(* Logix 5000 project; controller test vendor 1 type 14 code 151 rev 30.11; software revision 30.00 *)

TASK MainTask (continuous, watchdog 500 ms) : MainProgram

MODULES
   Local : vendor 1 type 14 code 151 (Compact 0, rev 30.11)
      Analog_IO : Embedded (Compact 2, rev 1.1, Output RPI 80 ms)
      Discrete_IO : Embedded (Compact 1, rev 3.1, Output RPI 20 ms)
      Counters : Embedded (Compact 3, rev 1.1, Output RPI 20 ms)
END_MODULES

PROGRAM MainProgram   (* main routine MainRoutine *)
VAR
   DI0 : ALIAS FOR Local:1:I.Data.0;
   DI1 : ALIAS FOR Local:1:I.Data.1;
   DI10 : ALIAS FOR Local:1:I.Data.10;
   DI11 : ALIAS FOR Local:1:I.Data.11;
   DI2 : ALIAS FOR Local:1:I.Data.2;
   DI3 : ALIAS FOR Local:1:I.Data.3;
   DI4 : ALIAS FOR Local:1:I.Data.4;
   DI5 : ALIAS FOR Local:1:I.Data.5;
   DI6 : ALIAS FOR Local:1:I.Data.6;
   DI61 : ALIAS FOR Local:1:I.Data.6;
   DI7 : ALIAS FOR Local:1:I.Data.7;
   DI8 : ALIAS FOR Local:1:I.Data.8;
   DI9 : ALIAS FOR Local:1:I.Data.9;
   DO0 : ALIAS FOR Local:1:O.Data.0;
   DO1 : ALIAS FOR Local:1:O.Data.1;
   DO10 : ALIAS FOR Local:1:O.Data.10;
   DO11 : ALIAS FOR Local:1:O.Data.11;
   DO2 : ALIAS FOR Local:1:O.Data.2;
   DO3 : ALIAS FOR Local:1:O.Data.3;
   DO4 : ALIAS FOR Local:1:O.Data.4;
   DO5 : ALIAS FOR Local:1:O.Data.5;
   DO6 : ALIAS FOR Local:1:O.Data.6;
   DO7 : ALIAS FOR Local:1:O.Data.7;
   DO8 : ALIAS FOR Local:1:O.Data.8;
   DO9 : ALIAS FOR Local:1:O.Data.9;
END_VAR

ROUTINE MainRoutine   (* ladder *)
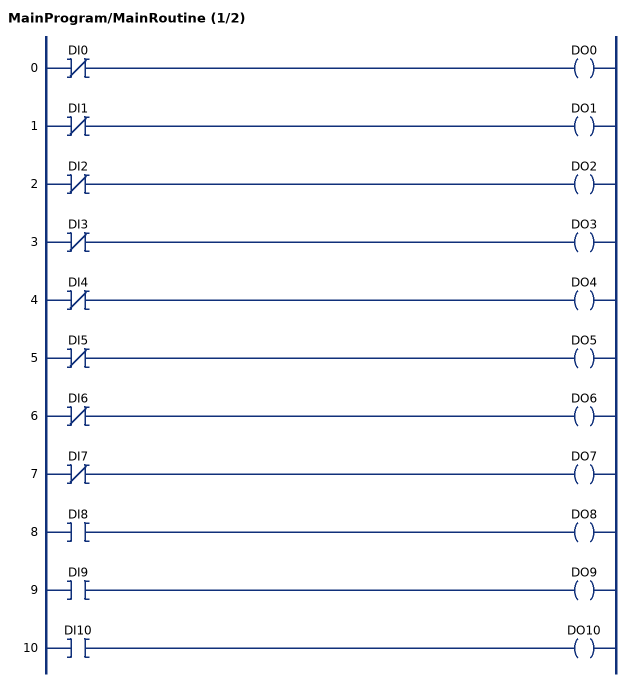
   0: XIO(DI0)OTE(DO0);
   1: XIO(DI1)OTE(DO1);
   2: XIO(DI2)OTE(DO2);
   3: XIO(DI3)OTE(DO3);
   4: XIO(DI4)OTE(DO4);
   5: XIO(DI5)OTE(DO5);
   6: XIO(DI6)OTE(DO6);
   7: XIO(DI7)OTE(DO7);
   8: XIC(DI8)OTE(DO8);
   9: XIC(DI9)OTE(DO9);
   10: XIC(DI10)OTE(DO10);
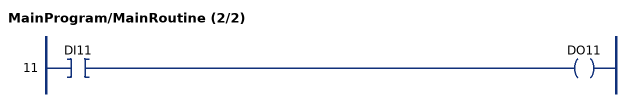
   11: XIC(DI11)OTE(DO11);
END_ROUTINE
END_PROGRAM
